Omron CX-Programmer project NewProject (CX-Programmer 9.75)

# PLC NewPLC1: CP1E E20

## Program NewProgram1 (cyclic task 0)

### Section Section1

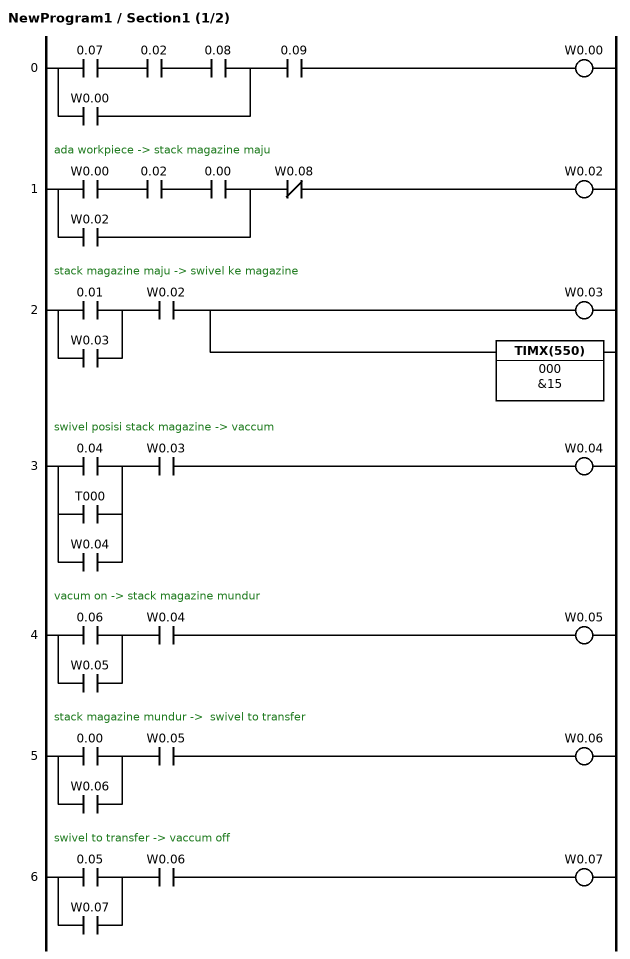
; rung 0
LD 0.07
AND 0.02
AND 0.08
OR W0.00
AND 0.09
OUT W0.00
; rung 1: ada workpiece -> stack magazine maju
LD W0.00
AND 0.02
AND 0.00
OR W0.02
ANDNOT W0.08
OUT W0.02
; rung 2: stack magazine maju -> swivel ke magazine
LD 0.01
OR W0.03
AND W0.02
OUT W0.03
TIMX(550) 000 &15
; rung 3: swivel posisi stack magazine -> vaccum
LD 0.04
OR T000
OR W0.04
AND W0.03
OUT W0.04
; rung 4: vacum on -> stack magazine mundur
LD 0.06
OR W0.05
AND W0.04
OUT W0.05
; rung 5: stack magazine mundur ->  swivel to transfer
LD 0.00
OR W0.06
AND W0.05
OUT W0.06
; rung 6: swivel to transfer -> vaccum off
LD 0.05
OR W0.07
AND W0.06
OUT W0.07

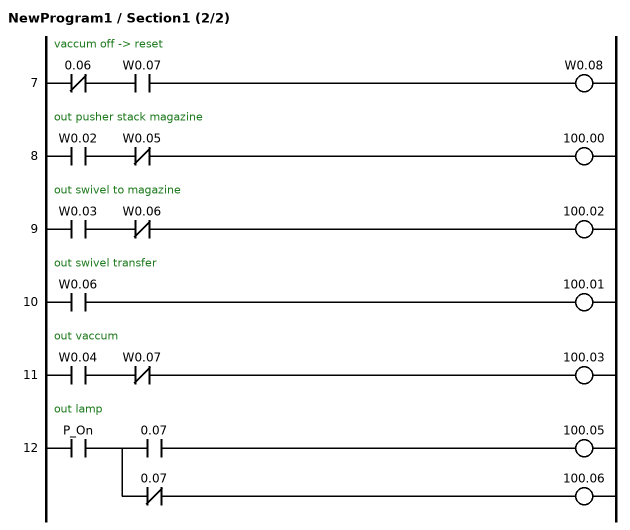
; rung 7: vaccum off -> reset
LDNOT 0.06
AND W0.07
OUT W0.08
; rung 8: out pusher stack magazine
LD W0.02
ANDNOT W0.05
OUT 100.00
; rung 9: out swivel to magazine
LD W0.03
ANDNOT W0.06
OUT 100.02
; rung 10: out swivel transfer
LD W0.06
OUT 100.01
; rung 11: out vaccum
LD W0.04
ANDNOT W0.07
OUT 100.03
; rung 12: out lamp
LD P_On
OUT TR0
AND 0.07
OUT 100.05
LD TR0
ANDNOT 0.07
OUT 100.06

### Section END
; rung 0
END(001)